INTERFACE ITF_EM_Labeller

END_INTERFACE

(* stored: Version 1.1.0.1, ProductVersion 3.1.4024.12
   Itf ITF_EM_Labeller: Id {69d47b9b-4851-45f7-bf20-2adb7572f65a} *)
